FUNCTION_BLOCK Ass_Openbox IMPLEMENTS ITF_AutoStructCommand
VAR_INPUT
END_VAR
VAR_OUTPUT
END_VAR
VAR
	strText	:STRING;
	i	:INT;
	MC_MoveAbsolute		: MC_MoveAbsolute;
	MC_Home				: MC_Home;
	_bProcessScan,_bInitialScan: BOOL;
	_bHalt , _bError,_bHaltPause: BOOL;
	nStep,nStt,nInitiStep	: INT;
	nNextStep		: INT;
	tmrClear		:TON;
	temp: DWORD;
	tmrloadIn,tmrloadIn2,tmrDelay: TON;
	wPunchcounter	:INT;
	_tmrT0: TON;
END_VAR

MC_Home(Axis:= Axis_BoxPullOut,bCalibrationCam := NOT Sen_AxisBoxORG);

IF NOT _bInitialScan THEN
	nInitiStep	:= 0;
END_IF

_bInitialScan:=FALSE;



IF NOT _bProcessScan THEN
	nNextStep	:= 0;
	nStep		:= 0;
END_IF

_bProcessScan	:=FALSE;

{warning 'add property implementation'}
PROPERTY Connect : STRING(50)
GET
END_GET
SET
END_SET
END_PROPERTY

METHOD INTERNAL Cyl_Safe : BOOL
VAR_INPUT
END_VAR
Cyl_Safe	:= Cyl_AxisBoxCatch.iOriginSensor AND Cyl_Axis90.iOriginSensor AND
				Cyl_AxisBottom.iOriginSensor AND Cyl_BoxSideBottom.iOriginSensor AND 	
				Cyl_BoxSidePitch.iOriginSensor	AND Cyl_BeltBottom.iOriginSensor ;
END_METHOD

{warning 'add property implementation'}
PROPERTY Error : BOOL
GET
END_GET
END_PROPERTY

{warning 'add method implementation '}
METHOD ErrorClear : BOOL
END_METHOD

{warning 'add method implementation '}
METHOD FB_init : BOOL
VAR_INPUT
	(* if TRUE, the retain variables are initialized (warm start / cold start)*)
	bInitRetains	: BOOL;
	(* if TRUE, the instance afterwards gets moved into the copy code (online change)*)
	bInCopyCode	: BOOL;
END_VAR
END_METHOD

METHOD HaltStepContiune : BOOL
nStep:= nNextStep;
END_METHOD

METHOD Initialization : BOOL
VAR_INPUT
	_Testmode	:BOOL;	//OOP Var
END_VAR
VAR
	bConfig: BOOL;
END_VAR
_bInitialScan	:= TRUE;
//初始化部屬 
//	IF Axis_BoxPullOut.Status.Error AND nInitiStep <> 100 THEN
//		nInitiStep:= 99;
//	END_IF
	
CASE nInitiStep OF
	0:
		_tmrT0(IN:=FALSE);
		strText:='ORG : Initial ';
		MC_Home.Execute:=FALSE;
		MC_MoveAbsolute(Axis:= Axis_BoxPullOut,Execute:=FALSE);
			
		Vacm_AxisCatchBox				:=FALSE;
		Cyl_AxisBoxCatch.qExtendCoil	:=FALSE;
		Cyl_Axis90.qExtendCoil			:=FALSE;
		Cyl_AxisBottom.qExtendCoil		:=FALSE;

		Vacm_Axis90						:=FALSE;
		Cyl_BoxSideBottom.qExtendCoil	:=FALSE;
		Cyl_BoxSidePitch.qExtendCoil	:=FALSE;
		
		Cyl_BeltBottom.qExtendCoil		:=FALSE;
		
		IF Cyl_Safe() THEN
			nInitiStep	:= 1;
		END_IF
	1:

	_tmrT0(IN:= NOT _tmrT0.Q ,PT:= T#1S);
	CASE Axis_BoxPullOut.Status.MotionState OF
		MC_AXISSTATE_UNDEFINED:
			;
		MC_AXISSTATE_DISABLED:
			IF Axis_BoxPullOut.Status.Error THEN
				Axis_BoxPullOut.Reset();
				ELSE
				Axis_BoxPullOut.ServoOn();
			END_IF;
		MC_AXISSTATE_STANDSTILL:
			;
		MC_AXISSTATE_ERRORSTOP:
			Axis_BoxPullOut.Reset();
		MC_AXISSTATE_CONTINOUSMOTION:
			Axis_BoxPullOut.Stop();
		MC_AXISSTATE_SYNCHRONIZEDMOTION	:
		;
	END_CASE
	
	IF Axis_BoxPullOut.Status.MotionState =MC_AXISSTATE_STANDSTILL THEN
		_tmrT0(IN:=FALSE);
		nInitiStep	:= 5;
	END_IF
	IF _tmrT0.Q THEN
		_tmrT0(IN:=FALSE);
		nInitiStep	:= 5;		
	END_IF

	5:
		bConfig			:=TRUE;
		IF NOT Axis_BoxPullOut.Status.StandStill THEN
			bConfig			:=FALSE;
			EventLogger.eEventType		:= 4;
			EventLogger.strEventText	:= 'BoxPullOutAxis Error ';	
			EventLogger();					
		END_IF
		
		IF bConfig THEN
			EventLogger.eEventType		:= 2;
			EventLogger.strEventText	:= 'BoxPull ORG Runing ';	
			EventLogger();
			_tmrT0(IN:= FALSE);
			nInitiStep:= nInitiStep + 5 ;
			strText:='ORG : Runing ';
			ELSE
			EventLogger.eEventType		:= 4;
			EventLogger.strEventText	:= 'Exceptions Cause interruptions!! ';	
			EventLogger();
			OP.bInitialSign		:=FALSE;
			OP.xInitialRuning	:=FALSE;
			nInitiStep := nInitiStep +100;	
			strText:='ORG : Failed ';
		END_IF	
		
	10:
		IF NOT Axis_BoxPullOut.Status.Homed THEN
			strText:='ORG : Runing ';
			nInitiStep	:= 16;
			ELSE
			strText:='ORG : Runing ';	
			nInitiStep	:= 17;
		END_IF;	
	//Axis Find Home
	16:
		MC_Home.Execute:=TRUE;
		IF MC_Home.Done THEN
			nInitiStep	:= 17;
		END_IF
		
	
	//Axis Go Abs SDANDBY Pos
	17:
		MC_MoveAbsolute(Axis:= Axis_BoxPullOut,Execute:=TRUE,Position:= RunParameter.Unboxing_PullOut,Velocity:= RunParameter.Unboxing_Velo);
			
		IF MC_MoveAbsolute.Done THEN
			MC_Home(Axis:= Axis_BoxPullOut,Execute:=FALSE);
			MC_MoveAbsolute(Axis:= Axis_BoxPullOut,Execute:=FALSE);	
			nInitiStep	:= 20;
		END_IF	
		
		
		
	//JobDone		
	20:
		strText:='ORG : Done ';
		Initialization	:= TRUE;	
	//Error step
	99:	
		IF Axis_BoxPullOut.DeviceErrorcode <> 0  THEN
			EventLogger.eEventType	:= E_EventType.Error;
			EventLogger.strEventText:= 'UnboxServo Driver Error';
			EventLogger.strEventText:= CONCAT(EventLogger.strEventText,WORD_TO_STRING(Axis_BoxPullOut.DeviceErrorcode));
			EventLogger();
		END_IF
		
		nInitiStep	:= 100;
END_CASE
END_METHOD

{warning 'add property implementation'}
PROPERTY NoEntry : BOOL
GET
END_GET
END_PROPERTY

{warning 'add method implementation '}
METHOD Pause : BOOL
END_METHOD

METHOD Process : BOOL		//OOP Return
VAR_INPUT
	bHlatMode	: BOOL;		//OOP Var
END_VAR
VAR
	_strTemp	:STRING[50];
END_VAR
_bProcessScan	:= TRUE;
//判斷 

IF _bError THEN
	strText	:= 'OpenBox:Error ';
	strText	:= CONCAT(Status,INT_TO_STRING(nStep));
END_IF;
//半自動模式
IF NOT bHlatMode  THEN
	nStep:= nNextStep;	
END_IF;

_bHaltPause	:= nStep<> nNextStep;
IF _bError OR _bHaltPause THEN
	RETURN;
END_IF

//主程序 
IF NOT _bHaltPause THEN
	tmrloadIn(in:= NOT tmrloadIn.q , PT:=RunParameter.Unboxing_DelayTime[0]);	
	IF tmrloadIn.Q THEN
		IF NOT Sen_BoxsideFeed THEN
			wPunchcounter	:= 	wPunchcounter + 1 ;
			Cyl_BoxSidePitch.qExtendCoil:= TRUE;
			ELSE
			wPunchcounter	:= 0;			
		END_IF
	END_IF;
	tmrloadIn2(IN:= Cyl_BoxSidePitch.iEndSensor ,PT:= T#1S);
	IF tmrloadIn2.q THEN
		Cyl_BoxSidePitch.qExtendCoil:= FALSE;			
	END_IF
	
	
	CASE nStep OF
		0:
			tmrDelay(IN:=FALSE);
			MC_MoveAbsolute(Axis:=Axis_BoxPullOut,Execute:=FALSE);
			IF Axis_BoxPullOut.Status.MotionState= MC_AXISSTATE_STANDSTILL AND Axis_BoxPullOut.Status.Homed THEN
				strText:= '';
				nNextStep	:= 10;
				nStep		:= 10;
				ELSE
				nNextStep	:= 100;
				nStep		:= 100;	
				strText:= '馬達狀態異常 ';			
			END_IF;
			
		10:
			MC_MoveAbsolute(Axis:= Axis_BoxPullOut,Execute:=TRUE,Position:= RunParameter.Unboxing_PullOut,Velocity:= RunParameter.Unboxing_Velo);
			IF MC_MoveAbsolute.Done THEN
				MC_MoveAbsolute(Axis:=Axis_BoxPullOut,Execute:=FALSE);
				nNextStep	:= 15;
			END_IF	
		15:
			Cyl_AxisBoxCatch.qExtendCoil	:= TRUE;
			IF Cyl_AxisBoxCatch.iEndSensor THEN
				nNextStep	:= 20;
			END_IF
		20:
			Vacm_AxisCatchBox:= TRUE;
			IF Sen_AxisBoxCatchVacumm THEN
				nNextStep	:= 21;
			END_IF
		21:
			Cyl_AxisBoxCatch.qExtendCoil	:= FALSE;	
			IF Cyl_AxisBoxCatch.iOriginSensor THEN
				nNextStep	:= 22;
			END_IF			
		22:
			Cyl_Axis90.qExtendCoil	:= TRUE;	
			tmrDelay(IN:= Cyl_Axis90.iEndSensor , pt:= T#1S);
			IF Cyl_Axis90.iEndSensor THEN
				tmrDelay(IN:=FALSE);
				nNextStep	:= 23;
			END_IF
		23:		
			Vacm_Axis90				:= TRUE;
			IF Sen_Axis90Vacumm THEN
				nNextStep	:= 24;
			END_IF
		24:
			Cyl_AxisBottom.qExtendCoil	:= TRUE;
			IF Cyl_AxisBottom.iEndSensor THEN
				nNextStep	:= 25;
			END_IF

		25:
			MC_MoveAbsolute(Axis:= Axis_BoxPullOut,Execute:=TRUE,Position:= RunParameter.Unboxing_PullOut+60,Velocity:= RunParameter.Unboxing_Velo);


			IF MC_MoveAbsolute.Done THEN
				MC_MoveAbsolute(Axis:=Axis_BoxPullOut,Execute:=FALSE);
				nNextStep	:= 26;
			END_IF
		26:
			Cyl_BeltBottom.qExtendCoil	:= TRUE;
			IF  Cyl_BeltBottom.iEndSensor THEN
				nNextStep	:= 27;
			END_IF		

		27:
			Cyl_BoxSideBottom.qExtendCoil	:= TRUE;
			IF Cyl_BoxSideBottom.iEndSensor THEN
				nNextStep	:= 28;
			END_IF

		28:
			tmrDelay(IN:=FALSE);
			strText:= 'Wait for Next St. ';	

			IF M_Sealing2.Connect = 'OpenBox In' THEN
				nNextStep	:= 30;
			END_IF
			
			IF NOT OP.xAutoMode THEN
				nNextStep	:= 30;
			END_IF
	
		30:
			//MC_MoveAbsolute(Axis:= Axis_BoxPullOut,Execute:=TRUE,Position:= RunParameter.Unboxing_LoadOut,Velocity:= RunParameter.Unboxing_Velo);
			MC_MoveAbsolute(Axis:= Axis_BoxPullOut,Execute:=TRUE,Position:= RunParameter.Unboxing_LoadOut,Velocity:= 100);

		IF Sen_BeltLoadIn THEN
				Cyl_BeltBottom.qExtendCoil		:= TRUE;
				Cyl_BoxSideBottom.qExtendCoil	:= FALSE;
				Vacm_AxisCatchBox				:=FALSE;
				//Cyl_AxisBottom.qExtendCoil		:= FALSE;
				Cyl_BeltBottom.qExtendCoil		:= FALSE;
				//Cyl_Axis90.qExtendCoil			:= FALSE;	
				Vacm_Axis90						:= FALSE;
			END_IF
			tmrDelay(IN:=MC_MoveAbsolute.Done,PT:=T#2S);
			IF tmrDelay.Q  THEN
				Cyl_BoxSideBottom.qExtendCoil	:= FALSE;
				Vacm_AxisCatchBox			:=FALSE;
				Cyl_AxisBottom.qExtendCoil	:= FALSE;
				Cyl_AxisBottom.qExtendCoil	:= FALSE;
				Cyl_BeltBottom.qExtendCoil	:= FALSE;
				Cyl_Axis90.qExtendCoil	:= FALSE;	
				Vacm_Axis90				:= FALSE;
				MC_MoveAbsolute(Axis:=Axis_BoxPullOut,Execute:=FALSE);
				nNextStep	:= 50;
			END_IF		

	

		50:
			IF OP.xAutoMode AND M_Sealing2.Connect = 'OpenBox In' THEN
				nNextStep	:= 0;
			END_IF
			;
	END_CASE
END_IF;

Process	:= nStep =50;
END_METHOD

PROPERTY Status : STRING(50)
GET
END_GET
END_PROPERTY

END_FUNCTION_BLOCK

(* stored: Version 1.1.0.1, ProductVersion 3.1.4026.18
   POU Ass_Openbox: Id {6fbfd320-f751-4f5c-aa0c-b173d550b2ff}, SpecialFunc None
   Property Connect: Id {f8a0cc84-e528-48fb-9909-0d076c8ed288}
   Get Get: Id {916ac29f-c4ba-414e-b515-aab1610a8f15}
   Set Set: Id {b4621454-94b4-4039-b20a-893c9648ac9d}
   Method Cyl_Safe: Id {7dd6f484-6ef4-4250-8a57-ff6fe0135fe9}
   Property Error: Id {99a50443-c8ff-44e1-be1d-7897cb57eb9c}
   Get Get: Id {546d74a7-10a9-4ddf-b2cf-c3b21f91dbbd}
   Method ErrorClear: Id {f5177dd6-d91c-416b-9996-3213b7f3eaf5}
   Method FB_init: Id {5c308be5-1d5e-4ea1-bbbe-6ed8bda94146}
   Method HaltStepContiune: Id {c273045f-2497-49da-9d86-8c8a24f4e1cd}
   Method Initialization: Id {d94725ae-728a-4d23-b958-9e593abe157c}
   Property NoEntry: Id {befa025c-d2f0-40e8-9b59-96ee3d462de7}
   Get Get: Id {f7bbb03f-72cd-41cc-86ee-ecaef34c9ca5}
   Method Pause: Id {ba2412fb-0b39-4975-9760-48b5002ca4b2}
   Method Process: Id {c66cbcd7-edc7-4b8f-8855-86abcab135c8}
   Property Status: Id {e31a4545-886a-4753-aeff-d91c2be66bdd}
   Get Get: Id {8ad3093b-77ce-46b2-8d36-ab7b614c243a} *)
